// TIA Portal V17 export
// export: Created 2022-02-03T14:45:13.4619293Z, ExportSetting WithDefaults, DisplayName Totally Integrated Automation Portal, DisplayVersion V17, DisplayName TIA Portal Openness, DisplayVersion V17, DisplayName TIA Portal Version Control Interface, DisplayVersion V17, DisplayName SINAMICS Startdrive Advanced, DisplayVersion V17, DisplayName SINAMICS Startdrive G130, G150, S120, S150, SINAMICS MV, S210, DisplayVersion V17, DisplayName SINAMICS Startdrive G110M, G120, G120C, G120D, G120P, G115D, DisplayVersion V17, DisplayName STEP 7 Professional, DisplayVersion V17, DisplayName STEP 7 Safety, DisplayVersion V17, DisplayName WinCC Advanced, DisplayVersion V17
DATA_BLOCK "ConveyorWeights_DB"   // DB7
VERSION : 0.1
// stored: Access Unpublished, AutoNumber true, DBAccessibleFromOPCUA true, DBAccessibleFromWebserver true, InstanceOfName ConveyorWeights, InstanceOfType FB
"ConveyorWeights"
   // VAR_INPUT
   //    weightSimulation : UInt;
   //    bLightBarrier : Bool;
   //    conveyorLeft : Bool;
   //    occupiedBay : Array["FIRSTBAY".."LASTBAY"] of Bool;
   // END_VAR
   // VAR_OUTPUT
   //    weightLightBarrier : UInt;
   //    weightBay : Array["FIRSTBAY".."LASTBAY"] of UInt;
   // END_VAR
   // VAR_IN_OUT
   //    weightConveyor : UInt;
   // END_VAR
   // VAR
   //    statOldbLightBarrier : Bool;
   //    statOldOccupiedBay : Array["FIRSTBAY".."LASTBAY"] of Bool;
   //    InstIEC_Timer1 { S7_SetPoint := 'True'} : TON_TIME;
   //    InstIEC_Timer2 { S7_SetPoint := 'True'} : TON_TIME;
   //    InstIEC_Timer3 { S7_SetPoint := 'True'} : TON_TIME;
   // END_VAR
BEGIN
END_DATA_BLOCK
